// TIA Portal V18 export
FUNCTION_BLOCK "FB_NG_Box_Control"   // FB5, SCL
{ S7_Optimized_Access := 'TRUE' }
// stored: MemoryReserve 1000, SetENOAutomatically false
   VAR_INPUT
      Button : Bool;
      MagnetSensor : Bool;
      LockedFB : Bool;
      UnlockedFB : Bool;
      AtSafePoint : Bool;
      Sensors : Array[1..15] of Bool;
   END_VAR
   VAR_OUTPUT
      PauseReq : Bool;
      UnlockCmd : Bool;
      LockCmd : Bool;
      CylinderOpen : Bool;
      CylinderClose : Bool;
      ButtonLight : Bool;
      Ready_1 : Bool;
      Ready_2 : Bool;
      Ready_3 : Bool;
      OpenFlag : Bool;
   END_VAR
   VAR
      State : Int := 99;
      BlinkTimer { S7_SetPoint := 'True'} : TON_TIME;
      BlinkBit : Bool;
      i : Int;
      buttontriggered { S7_SetPoint := 'True'} : R_TRIG;
      c : Int;
   END_VAR
BEGIN
   // 1. POSITION CHECK (Ready_1..3) - TRUE = at least one position in the row is FREE
   // 1. KONTROLA POZÍCIÍ – TRUE = aspoň jedna pozícia v rade je VOĽNÁ
   // 1. 位置检测 – TRUE = 该行中至少有一个位置是空的

   // LINE #1  .... 5 POSITIONS
   // EN: Line 1 checks sensors 1–5 (row 1)
   // SK: Riadok 1 kontroluje senzory 1–5 (riadok 1)
   // CN: 第1行检测传感器1–5（第1排）
   #Ready_1 := FALSE;
   FOR #i := 1 TO 5 DO
     IF NOT #Sensors[#i] THEN
       #Ready_1 := TRUE;
     END_IF;
   END_FOR;

   // LINE #2  .... 5 POSITIONS
   // EN: Line 2 checks sensors 6–10 (row 2)
   // SK: Riadok 2 kontroluje senzory 6–10 (riadok 2)
   // CN: 第2行检测传感器6–10（第2排）
   #Ready_2 := FALSE;
   FOR #i := 6 TO 10 DO
     IF NOT #Sensors[#i] THEN
       #Ready_2 := TRUE;
     END_IF;
   END_FOR;

   // LINE #3  .... 5 POSITIONS
   // EN: Line 3 checks sensors 11–15 (row 3)
   // SK: Riadok 3 kontroluje senzory 11–15 (riadok 3)
   // CN: 第3行检测传感器11–15（第3排）
   #Ready_3 := FALSE;
   FOR #i := 11 TO 15 DO
     IF NOT #Sensors[#i] THEN
       #Ready_3 := TRUE;
     END_IF;
   END_FOR;


   // 2. BLINKING / BUTTON FEEDBACK
   // EN: Blink signal taken from system clock (0.4s)
   // SK: Blikanie je odvodené zo systémového hodinového bitu (0,4 s)
   // CN: 闪烁信号来自系统时钟位（0.4秒）
   #BlinkBit := "ClockMemory0.4s";

   // EN: Rising-edge detection of the button
   // SK: Detekcia nábežnej hrany tlačidla
   // CN: 按钮上升沿检测
   #buttontriggered(CLK := #Button);


   // 3. DOOR STATE MACHINE
   // EN: Main state machine controlling door, lock and cylinder
   // SK: Hlavný stavový automat pre dvere, zámok a valec
   // CN: 门、锁和气缸的主状态机
   CASE #State OF

     99: // INITIALIZATION
       // EN: Decision after PLC start
       // SK: Rozhodnutie po štarte PLC
       // CN: PLC 启动后的状态判断
       IF #MagnetSensor AND #LockedFB THEN
         #State := 0;   // EN: Closed & locked → IDLE
         // SK: Zavreté a zamknuté → IDLE
         // CN: 已关闭并锁定 → 空闲状态
       ELSIF #MagnetSensor AND NOT #LockedFB THEN
         #State := 40;  // EN: Closed but unlocked → wait for confirmation
         // SK: Zavreté, ale odomknuté → čakať na potvrdenie
         // CN: 门已关但未上锁 → 等待确认
       ELSE
         #State := 30;  // EN: Door physically open → OPEN state
         // SK: Dvere fyzicky otvorené → OPEN stav
         // CN: 门处于打开状态 → OPEN
       END_IF;

     0:  // IDLE
       // EN: Normal operation, sequence running
       // SK: Normálna prevádzka, sekvencia beží
       // CN: 正常运行，工序执行中
       #PauseReq := FALSE;
       #UnlockCmd := FALSE;
       #LockCmd := TRUE;
       #CylinderOpen := FALSE;
       #CylinderClose := TRUE;
       #ButtonLight := TRUE;
       #OpenFlag := FALSE;
       IF #buttontriggered.Q THEN
         #State := 10;
       END_IF;

     10: // REQUEST
       // EN: Button pressed, waiting for safe point (Step 111)
       // SK: Tlačidlo stlačené, čaká sa na bezpečný bod (Krok 111)
       // CN: 按钮按下，等待安全点（步骤111）
       #PauseReq := TRUE;
       #ButtonLight := #BlinkBit;
       IF #AtSafePoint THEN
         #State := 20;
       END_IF;

     20: // SAFE
       // EN: Sequence stopped, unlocking door and opening cylinder
       // SK: Sekvencia stojí, odomykáme dvere a otvárame valec
       // CN: 工序停止，解锁门并打开气缸
       #PauseReq := TRUE;
       #UnlockCmd := TRUE;
       #LockCmd := FALSE;
       #ButtonLight := #BlinkBit;
       IF #UnlockedFB THEN
         #CylinderOpen := TRUE;
         #CylinderClose := FALSE;
         #State := 30;
       END_IF;

     30: // OPEN
       // EN: Door open, operator access
       // SK: Dvere otvorené, obsluha má prístup
       // CN: 门已打开，操作员可进入
       #PauseReq := TRUE;
       #ButtonLight := FALSE;
       #OpenFlag := TRUE;
       #UnlockCmd := TRUE;
       #LockCmd := FALSE;
       #CylinderOpen := TRUE;
       #CylinderClose := FALSE;
       IF #MagnetSensor THEN
         #State := 40;
       END_IF;

     40: // CONFIRM
       // EN: Door closed, waiting for operator confirmation
       // SK: Dvere zatvorené, čaká sa na potvrdenie obsluhou
       // CN: 门已关闭，等待人工确认
       #PauseReq := TRUE;
       #ButtonLight := #BlinkBit;
       #OpenFlag := TRUE;
       #UnlockCmd := TRUE;
       #LockCmd := FALSE;
       #CylinderOpen := TRUE;
       #CylinderClose := FALSE;
       IF NOT #MagnetSensor THEN
         #State := 30;
       ELSIF #buttontriggered.Q THEN
         #State := 50;
       END_IF;

     50: // LOCKING
       // EN: Locking door and returning cylinder
       // SK: Zamykáme dvere a vraciame valec
       // CN: 锁门并回收气缸
       #PauseReq := TRUE;
       #CylinderOpen := FALSE;
       #CylinderClose := TRUE;
       #UnlockCmd := FALSE;
       #LockCmd := TRUE;
       IF #LockedFB THEN
         #PauseReq := FALSE; // EN: Release Step 111, sequence continues
         // SK: Uvoľní sa Krok 111, sekvencia pokračuje
         // CN: 释放步骤111，工序继续
         #State := 0;
       END_IF;

   END_CASE;


   // EN: Test lamp function from system diagnostics
   // SK: Testovacia funkcia lampy zo systémovej diagnostiky
   // CN: 系统诊断用的灯测试功能
   IF "Station_Sys".Cmd.TestLamp THEN
     #ButtonLight := TRUE;
   END_IF;
END_FUNCTION_BLOCK
